FUNCTION_BLOCK A2X_2X_TO_BOOL (* Composite FB for convert A2X to 2 BOOLS *)
  (* Standard: 61499-2; Description: Copyright (c) 2024 HR Agrartechnik GmbH This program and the accompanying materials are made available under the terms of the Eclipse Public License 2.0 which is available at https://www.eclipse.org/legal/epl-2.0/ SPDX-License-Identifier: EPL-2.0 *)
  (* Version 1.0, 2024-04-24, Franz Höpfinger, HR Agrartechnik GmbH *)
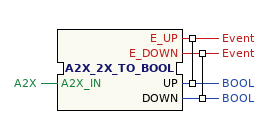
  EVENT_OUTPUT
    E_UP WITH UP; (* UP *)
    E_DOWN WITH DOWN; (* DOWN *)
  END_EVENT
  VAR_OUTPUT
    UP : BOOL; (* TRUE = forward, up, right, clockwise *)
    DOWN : BOOL; (* TRUE = backward, down, left, counter-clockwise *)
  END_VAR
  SOCKETS
    A2X_IN : A2X; (* Adapter Input *)
  END_SOCKETS
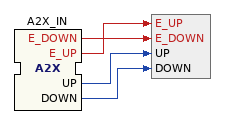
  EVENT_CONNECTIONS
    A2X_IN.E_DOWN TO E_DOWN;
    A2X_IN.E_UP TO E_UP;
  END_CONNECTIONS
  DATA_CONNECTIONS
    A2X_IN.UP TO UP;
    A2X_IN.DOWN TO DOWN;
  END_CONNECTIONS
END_FUNCTION_BLOCK
